{attribute 'GeneratedUsingTerminal: EL6784-0000-0016'}
{attribute addProperty BoxType "EL6784-0000-0016"}
{attribute addProperty Id "StatusAT %I*Status_07D3AAF62InputsEMPTY_STRUCTURE0ControlAT %Q*Control_DAFD38E02OutputsEMPTY_STRUCTURE0WcStateAT %I*WcState_9091E0EB2InfoDataAT %I*InfoData_94A18F5E2"}
{attribute addProperty CRC "2439747241"}
{attribute addProperty Size "8"}
TYPE EL6784_916B96A9 EXTENDS EtcSlaveTerminalBase_947E5A46 :
STRUCT
	{attribute addProperty Name "Status"}
	Status : Status_07D3AAF6;
	{attribute addProperty Name "Inputs"}
	Inputs : EMPTY_STRUCTURE;
	{attribute addProperty Name "Control"}
	Control : Control_DAFD38E0;
	{attribute addProperty Name "Outputs"}
	Outputs : EMPTY_STRUCTURE;
	{attribute addProperty Name "WcState"}
	WcState : WcState_9091E0EB;
	{attribute addProperty Name "InfoData"}
	InfoData : InfoData_94A18F5E;
END_STRUCT
END_TYPE

(* stored: Version 1.2.0.0, ProductVersion 3.1.4024.9
   DUT EL6784_916B96A9: Id {3e981cc0-5434-44ac-8aae-a7cecc75a747} *)
